// TIA Portal V19 export
TYPE "PPrf_Data"
// stored: Access Published
   STRUCT
      Header { S7_SetPoint := 'True'} : "Prg_Header";
      GeneralData { S7_SetPoint := 'True'} : "PPrf_Generic";
      SetUp { S7_SetPoint := 'True'} : "PPrf_SetUp";
      A01_CoilHandling { S7_SetPoint := 'True'} : "PPrf_CoilHandlig";
      A02_1_PartsCutting { S7_SetPoint := 'True'} : "PPrf_A02_S1_PartsCutting";
      A0301_A0302 { S7_SetPoint := 'True'} : "PPrf_A0301_0302_Assemblaggio";
      A0303_A0304 { S7_SetPoint := 'True'} : "PPrf_A0304_0304_Scarico";
   END_STRUCT;
END_TYPE
